(* PLC project Portifolio 1 .project, CODESYS CODESYS V3.5 SP21 Patch 4 *)
(* stored: creationDateTime 2026-02-13T15:16:45.32497, modificationDateTime 2026-02-13T15:00:39.8619068 *)

PROGRAM PRG_MotorControl
  VAR
    xToggleButton : BOOL;  (* Single button to Start/Stop (NO) *)
    xEmergencyStop_NC : BOOL := TRUE;  (* Emergency Stop (NC - TRUE is healthy) *)
    xThermalOK_NC : BOOL := TRUE;  (* Thermal Protection (NC - TRUE is healthy) *)
    fbButtonEdge : R_TRIG;  (* Edge detector to prevent multiple toggles *)
    xMotorState : BOOL;  (* Internal memory (Latch) for motor status *)
    xMotorCommand : BOOL;  (* Output to the Motor (Green Light) *)
    xEmergencyAlarmLight : BOOL;  (* Output to the Emergency Alarm (Red Light) *)
    xThermalAlarmLight : BOOL;  (* Output to the Thermal Alarm (Yellow Light) *)
  END_VAR

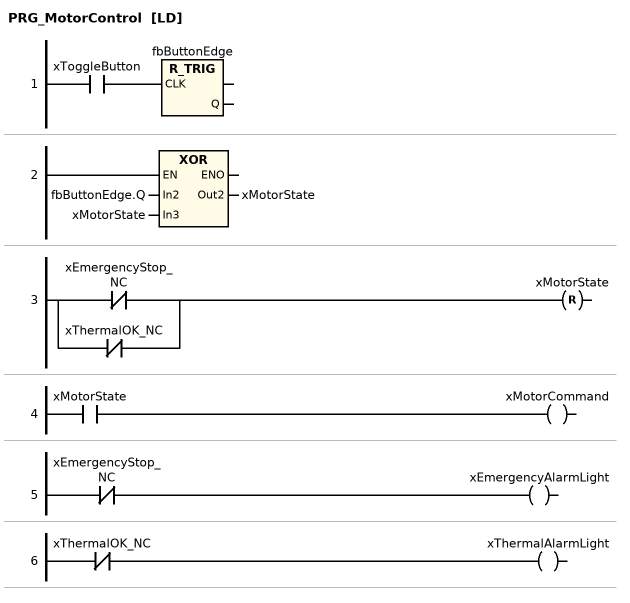
(* LD diagram, written out as Structured Text *)

fbButtonEdge(CLK := xToggleButton);

xMotorState := fbButtonEdge.Q XOR xMotorState;

IF NOT xEmergencyStop_NC OR NOT xThermalOK_NC THEN xMotorState := FALSE; END_IF;

xMotorCommand := xMotorState;

xEmergencyAlarmLight := NOT xEmergencyStop_NC;

xThermalAlarmLight := NOT xThermalOK_NC;
END_PROGRAM

PROGRAM PRG_MotorControl_ST
  VAR
    xToggleButton : BOOL;  (* Single button to Start/Stop (NO) *)
    xEmergencyStop_NC : BOOL := TRUE;  (* Emergency Stop (NC - TRUE is healthy) *)
    xThermalOK_NC : BOOL := TRUE;  (* Thermal Protection (NC - TRUE is healthy) *)
    fbButtonEdge : R_TRIG;  (* Edge detector to prevent multiple toggles *)
    xMotorState : BOOL;  (* Internal memory (Latch) for motor status *)
    xMotorCommand : BOOL;  (* Output to the Motor (Green Light) *)
    xEmergencyAlarmLight : BOOL;  (* Output to the Emergency Alarm (Red Light) *)
    xThermalAlarmLight : BOOL;  (* Output to the Thermal Alarm (Yellow Light) *)
  END_VAR

                  // ==============================================================================
// 1. EDGE DETECTION | DETECÇÃO DE BORDA
// EN: Detects the rising edge of the toggle button to prevent multiple triggers.
// PT: Detecta a borda de subida do botão para evitar múltiplos acionamentos.
// ==============================================================================
fbButtonEdge(CLK := xToggleButton);

// ==============================================================================
// 2. COMMAND LOGIC | LÓGICA DE COMANDO (Toggle via XOR)
// EN: Inverts the motor state securely at every single button click.
// PT: Inverte o estado do motor de forma segura a cada clique do operador.
// ==============================================================================
xMotorState := fbButtonEdge.Q XOR xMotorState;

// ==============================================================================
// 3. SAFETY INTERLOCKS | INTERTRAVAMENTOS DE SEGURANÇA (Fail-Safe)
// EN: If Emergency (FALSE) OR Thermal (FALSE), stop the motor. Priority to Reset.
// PT: Se Emergência (FALSE) OU Térmico (FALSE), desliga o motor. Prioridade ao Reset.
// ==============================================================================
IF NOT xEmergencyStop_NC OR NOT xThermalOK_NC THEN
    xMotorState := FALSE;
END_IF;

// ==============================================================================
// 4. OUTPUT MAPPING | MAPEAMENTO DAS SAÍDAS (HMI Indicators)
// EN: Map the internal states to the physical outputs and HMI lamps.
// PT: Mapeia os estados internos para as saídas físicas e lâmpadas da tela.
// ==============================================================================
xMotorCommand        := xMotorState;           // Green Light | Luz Verde
xEmergencyAlarmLight := NOT xEmergencyStop_NC; // Red Light   | Luz Vermelha
xThermalAlarmLight   := NOT xThermalOK_NC;     // Yellow Light| Luz Amarela
                
END_PROGRAM

CONFIGURATION Application
  RESOURCE Application ON PLC
    TASK MainTask(INTERVAL := T#20ms, PRIORITY := 1);
    TASK VISU_TASK(INTERVAL := T#100ms, PRIORITY := 31);
    PROGRAM PRG_MotorControl WITH MainTask : PRG_MotorControl;
    PROGRAM VisuElems.Visu_Prg WITH VISU_TASK : VisuElems.Visu_Prg;
  END_RESOURCE
END_CONFIGURATION
